// TIA Portal V20 export
FUNCTION_BLOCK "Simulation"   // FB147, LAD
// stored: MemoryReserve 100, Namespace Unit1.Em6, SetENOAutomatically false
   VAR
      Simulation_addon_Instance { S7_SetPoint := 'True'} : "Simulation_addon";
      statPulse { S7_SetPoint := 'True'} : Bool;
      statPulse_1 { S7_SetPoint := 'True'} : Bool;
      statSimulationVisionData : DInt;
      IEC_Timer_0_Instance { S7_SetPoint := 'True'} : TON_TIME;
      IEC_Timer_0_Instance_1 { S7_SetPoint := 'True'} : TON_TIME;
   END_VAR
   VAR_TEMP   // added for the SCL form of the ladder/FBD networks
      _w1 : Bool;
      _w2 : Bool;
      _w3 : Bool;
      _w4 : Bool;
   END_VAR
BEGIN

REGION Network 1: cmVisionPusherSupportUpDown
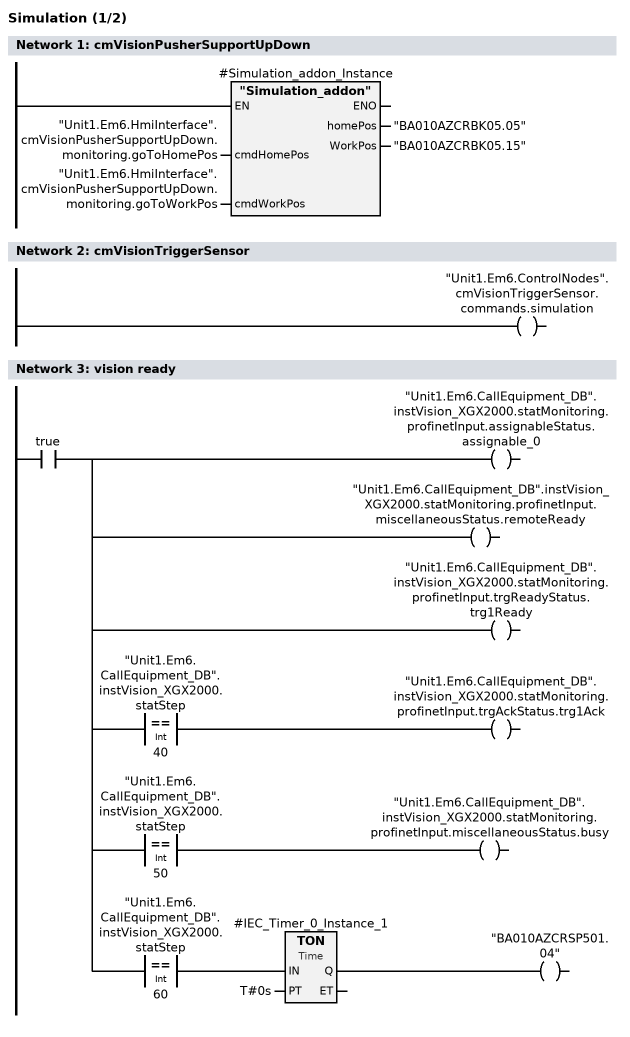
   RUNG wire#powerrail
      #Simulation_addon_Instance(cmdHomePos := "Unit1.Em6.HmiInterface".cmVisionPusherSupportUpDown.monitoring.goToHomePos, cmdWorkPos := "Unit1.Em6.HmiInterface".cmVisionPusherSupportUpDown.monitoring.goToWorkPos, homePos => "BA010AZCRBK05.05", WorkPos => "BA010AZCRBK05.15")
   END_RUNG
   // the same network as SCL:
   #Simulation_addon_Instance(cmdHomePos := "Unit1.Em6.HmiInterface".cmVisionPusherSupportUpDown.monitoring.goToHomePos,   // "Simulation_addon"
                           cmdWorkPos := "Unit1.Em6.HmiInterface".cmVisionPusherSupportUpDown.monitoring.goToWorkPos,
                           homePos => "BA010AZCRBK05.05",
                           WorkPos => "BA010AZCRBK05.15");
END_REGION

REGION Network 2: cmVisionTriggerSensor
   RUNG wire#powerrail
      Coil( "Unit1.Em6.ControlNodes".cmVisionTriggerSensor.commands.simulation )
   END_RUNG
   // the same network as SCL:
   "Unit1.Em6.ControlNodes".cmVisionTriggerSensor.commands.simulation := TRUE;
END_REGION

REGION Network 3: vision ready
   RUNG wire#powerrail
      Contact( true )
      wire#w1
      Coil( "Unit1.Em6.CallEquipment_DB".instVision_XGX2000.statMonitoring.profinetInput.assignableStatus.assignable_0 )
   END_RUNG
   RUNG wire#w1
      Coil( "Unit1.Em6.CallEquipment_DB".instVision_XGX2000.statMonitoring.profinetInput.miscellaneousStatus.remoteReady )
   END_RUNG
   RUNG wire#w1
      Coil( "Unit1.Em6.CallEquipment_DB".instVision_XGX2000.statMonitoring.profinetInput.trgReadyStatus.trg1Ready )
   END_RUNG
   RUNG wire#w1
      { S7_Templates := "SrcType := Int" } EQ_Contact(in1 := "Unit1.Em6.CallEquipment_DB".instVision_XGX2000.statStep, in2 := 40)
      Coil( "Unit1.Em6.CallEquipment_DB".instVision_XGX2000.statMonitoring.profinetInput.trgAckStatus.trg1Ack )
   END_RUNG
   RUNG wire#w1
      { S7_Templates := "SrcType := Int" } EQ_Contact(in1 := "Unit1.Em6.CallEquipment_DB".instVision_XGX2000.statStep, in2 := 50)
      Coil( "Unit1.Em6.CallEquipment_DB".instVision_XGX2000.statMonitoring.profinetInput.miscellaneousStatus.busy )
   END_RUNG
   RUNG wire#w1
      { S7_Templates := "SrcType := Int" } EQ_Contact(in1 := "Unit1.Em6.CallEquipment_DB".instVision_XGX2000.statStep, in2 := 60)
      { S7_Templates := "time_type := Time" } #IEC_Timer_0_Instance_1.TON(pt := T#0s, et =>)
      Coil( "BA010AZCRSP501.04" )
   END_RUNG
   // the same network as SCL:
   "Unit1.Em6.CallEquipment_DB".instVision_XGX2000.statMonitoring.profinetInput.assignableStatus.assignable_0 := true;
   "Unit1.Em6.CallEquipment_DB".instVision_XGX2000.statMonitoring.profinetInput.miscellaneousStatus.remoteReady := true;
   "Unit1.Em6.CallEquipment_DB".instVision_XGX2000.statMonitoring.profinetInput.trgReadyStatus.trg1Ready := true;
   "Unit1.Em6.CallEquipment_DB".instVision_XGX2000.statMonitoring.profinetInput.trgAckStatus.trg1Ack := true AND ("Unit1.Em6.CallEquipment_DB".instVision_XGX2000.statStep = 40);
   "Unit1.Em6.CallEquipment_DB".instVision_XGX2000.statMonitoring.profinetInput.miscellaneousStatus.busy := true AND ("Unit1.Em6.CallEquipment_DB".instVision_XGX2000.statStep = 50);
   #IEC_Timer_0_Instance_1(IN := true AND ("Unit1.Em6.CallEquipment_DB".instVision_XGX2000.statStep = 60),   // TON
                           PT := T#0s);
   "BA010AZCRSP501.04" := #IEC_Timer_0_Instance_1.Q;
END_REGION

REGION Network 4: Qr Reader
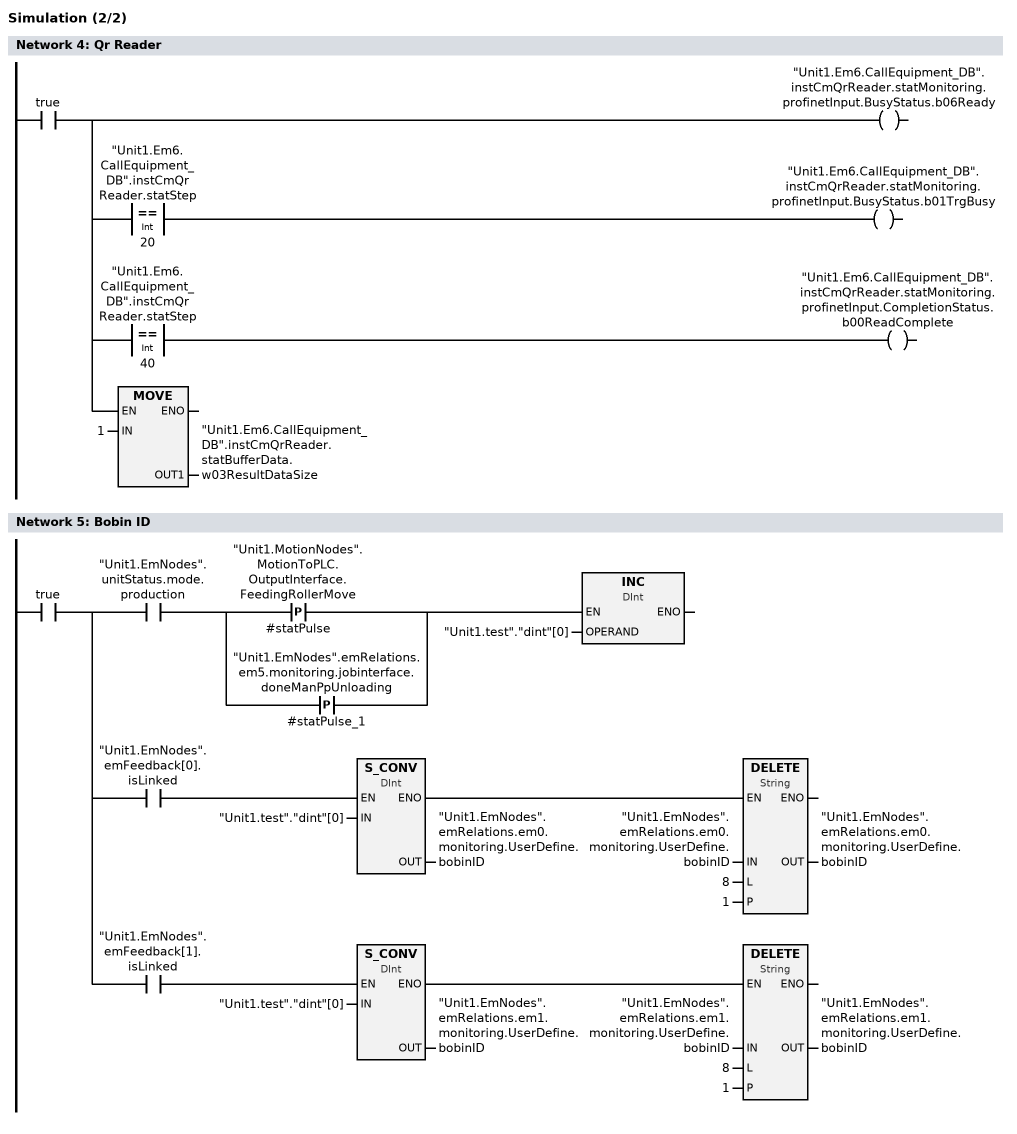
   RUNG wire#powerrail
      Contact( true )
      wire#w1
      Coil( "Unit1.Em6.CallEquipment_DB".instCmQrReader.statMonitoring.profinetInput.BusyStatus.b06Ready )
   END_RUNG
   RUNG wire#w1
      { S7_Templates := "SrcType := Int" } EQ_Contact(in1 := "Unit1.Em6.CallEquipment_DB".instCmQrReader.statStep, in2 := 20)
      Coil( "Unit1.Em6.CallEquipment_DB".instCmQrReader.statMonitoring.profinetInput.BusyStatus.b01TrgBusy )
   END_RUNG
   RUNG wire#w1
      { S7_Templates := "SrcType := Int" } EQ_Contact(in1 := "Unit1.Em6.CallEquipment_DB".instCmQrReader.statStep, in2 := 40)
      Coil( "Unit1.Em6.CallEquipment_DB".instCmQrReader.statMonitoring.profinetInput.CompletionStatus.b00ReadComplete )
   END_RUNG
   RUNG wire#w1
      Move(in := 1, out1 => "Unit1.Em6.CallEquipment_DB".instCmQrReader.statBufferData.w03ResultDataSize)
   END_RUNG
   // the same network as SCL:
   "Unit1.Em6.CallEquipment_DB".instCmQrReader.statMonitoring.profinetInput.BusyStatus.b06Ready := true;
   "Unit1.Em6.CallEquipment_DB".instCmQrReader.statMonitoring.profinetInput.BusyStatus.b01TrgBusy := true AND ("Unit1.Em6.CallEquipment_DB".instCmQrReader.statStep = 20);
   "Unit1.Em6.CallEquipment_DB".instCmQrReader.statMonitoring.profinetInput.CompletionStatus.b00ReadComplete := true AND ("Unit1.Em6.CallEquipment_DB".instCmQrReader.statStep = 40);
   IF true THEN "Unit1.Em6.CallEquipment_DB".instCmQrReader.statBufferData.w03ResultDataSize := 1; END_IF;
END_REGION

REGION Network 5: Bobin ID
   RUNG wire#powerrail
      Contact( true )
      wire#w1
      Contact( "Unit1.EmNodes".unitStatus.mode.production )
      wire#w2
      P_Contact(operand := "Unit1.MotionNodes".MotionToPLC.OutputInterface.FeedingRollerMove, bit := #statPulse)
      wire#w3
      { S7_Templates := "DestType := DInt" } Inc( "Unit1.test"."dint"[0] )
   END_RUNG
   RUNG wire#w2
      P_Contact(operand := "Unit1.EmNodes".emRelations.em5.monitoring.jobinterface.doneManPpUnloading, bit := #statPulse_1)
   END_RUNG wire#w3
   RUNG wire#w1
      Contact( "Unit1.EmNodes".emFeedback[0].isLinked )
      { S7_Templates := "[src_type := DInt, dest_type := String]" } S_CONV(IN := "Unit1.test"."dint"[0], OUT => "Unit1.EmNodes".emRelations.em0.monitoring.UserDefine.bobinID)
      { S7_Templates := "str_type := String" } DELETE(IN := "Unit1.EmNodes".emRelations.em0.monitoring.UserDefine.bobinID, L := 8, P := 1, OUT => "Unit1.EmNodes".emRelations.em0.monitoring.UserDefine.bobinID)
   END_RUNG
   RUNG wire#w1
      Contact( "Unit1.EmNodes".emFeedback[1].isLinked )
      { S7_Templates := "[src_type := DInt, dest_type := String]" } S_CONV(IN := "Unit1.test"."dint"[0], OUT => "Unit1.EmNodes".emRelations.em1.monitoring.UserDefine.bobinID)
      { S7_Templates := "str_type := String" } DELETE(IN := "Unit1.EmNodes".emRelations.em1.monitoring.UserDefine.bobinID, L := 8, P := 1, OUT => "Unit1.EmNodes".emRelations.em1.monitoring.UserDefine.bobinID)
   END_RUNG
   // the same network as SCL:
   #_w1 := true AND "Unit1.EmNodes".unitStatus.mode.production AND "Unit1.MotionNodes".MotionToPLC.OutputInterface.FeedingRollerMove AND NOT #statPulse;   // rising edge of "Unit1.MotionNodes".MotionToPLC.OutputInterface.FeedingRollerMove
   #statPulse := "Unit1.MotionNodes".MotionToPLC.OutputInterface.FeedingRollerMove;
   #_w2 := true AND "Unit1.EmNodes".unitStatus.mode.production AND "Unit1.EmNodes".emRelations.em5.monitoring.jobinterface.doneManPpUnloading AND NOT #statPulse_1;   // rising edge of "Unit1.EmNodes".emRelations.em5.monitoring.jobinterface.doneManPpUnloading
   #statPulse_1 := "Unit1.EmNodes".emRelations.em5.monitoring.jobinterface.doneManPpUnloading;
   IF #_w1 OR #_w2 THEN "Unit1.test"."dint"[0] := "Unit1.test"."dint"[0] + 1; END_IF;
   S_CONV(EN := true AND "Unit1.EmNodes".emFeedback[0].isLinked,
          IN := "Unit1.test"."dint"[0],
          OUT => "Unit1.EmNodes".emRelations.em0.monitoring.UserDefine.bobinID,
          ENO => #_w3);
   IF #_w3 THEN
       DELETE(IN := "Unit1.EmNodes".emRelations.em0.monitoring.UserDefine.bobinID,
              L := 8,
              P := 1,
              OUT => "Unit1.EmNodes".emRelations.em0.monitoring.UserDefine.bobinID);
   END_IF;
   S_CONV(EN := true AND "Unit1.EmNodes".emFeedback[1].isLinked,
          IN := "Unit1.test"."dint"[0],
          OUT => "Unit1.EmNodes".emRelations.em1.monitoring.UserDefine.bobinID,
          ENO => #_w4);
   IF #_w4 THEN
       DELETE(IN := "Unit1.EmNodes".emRelations.em1.monitoring.UserDefine.bobinID,
              L := 8,
              P := 1,
              OUT => "Unit1.EmNodes".emRelations.em1.monitoring.UserDefine.bobinID);
   END_IF;
END_REGION
END_FUNCTION_BLOCK
